PROGRAM MAIN
VAR
  nTest: INT;
  sTest: STRING;
END_VAR

END_PROGRAM

(* stored: Version 1.1.0.1, ProductVersion 3.1.4024.2
   POU MAIN: Id {c2b5ef02-c814-43e4-afb8-0f2b009686dc}, SpecialFunc None *)
